FUNCTION_BLOCK F_CONCAT_DT (* concatenation to DATE_AND_TIME *)
  (* Standard: 61131-3; Classification: standard character and string function; Description: Copyright (c) 2013 TU Wien ACIN and others. This program and the accompanying materials are made available under the terms of the Eclipse Public License 2.0 which is available at https://www.eclipse.org/legal/epl-2.0/ SPDX-License-Identifier: EPL-2.0 Some portions generated by Gemini CLI *)
  (* Version 1.0, 2026-01-31, Franz Höpfinger, HR Agrartechnik GmbH, F_CONCAT_DT copied from F_CONCAT and implemented according IEC 61131-3 *)
  PACKAGE iec61131::charString;
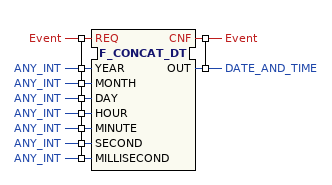
  EVENT_INPUT
    REQ WITH YEAR, MONTH, DAY, HOUR, MINUTE, SECOND, MILLISECOND; (* Service Request *)
  END_EVENT
  EVENT_OUTPUT
    CNF WITH OUT; (* Confirmation of Requested Service *)
  END_EVENT
  VAR_INPUT
    YEAR : ANY_INT; (* Year *)
    MONTH : ANY_INT; (* Month *)
    DAY : ANY_INT; (* Day *)
    HOUR : ANY_INT; (* Hour *)
    MINUTE : ANY_INT; (* Minute *)
    SECOND : ANY_INT; (* Second *)
    MILLISECOND : ANY_INT; (* Millisecond *)
  END_VAR
  VAR_OUTPUT
    OUT : DATE_AND_TIME; (* Resulting DATE_AND_TIME *)
  END_VAR
  EC_STATES
    REQ : REQ -> CNF;
  END_STATES
  ALGORITHM REQ IN ST:
OUT := CONCAT_DT(YEAR, MONTH, DAY, HOUR, MINUTE, SECOND, MILLISECOND);
  END_ALGORITHM
END_FUNCTION_BLOCK
